// LS Electric XG5000 project: OR
// PLC LSPLC
// module base 0 slot 0: 입출력 모듈:XBC-DR30S (DC 24V 입력 18점, 릴레이 출력 12점)

PROGRAM ORTEST (task: 스캔 프로그램)

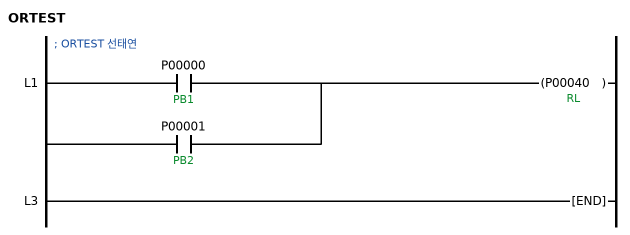
// ORTEST 선태연
; L1
LOAD      P00000	// PB1
OR        P00001	// PB2
OUT       P00040	// RL
; L3
END